(* PLC project BlogProject.project, CODESYS CODESYS V3.5 SP14 Patch 3 *)
(* stored: creationDateTime 2021-10-07T21:03:08.9474637, modificationDateTime 2021-10-07T20:40:20.1109198 *)

TYPE udtTransition : STRUCT
  eCurrentState : enumState;
  mcEvent_1 : itfEvent;
  mcEvent_2 : itfEvent;
  mcAction_1 : itfAction;
  mcAction_2 : itfAction;
  eNextStage : enumState;
END_STRUCT;
END_TYPE
